TYPE elementStatus :
(
    Bad := 0,
    Timeout := 1,
	Unknown := 11,
    Good := 12
);
END_TYPE

(* stored: Version 1.1.0.1, ProductVersion 3.1.0.36
   DUT elementStatus: Id {b682ee42-3264-4a62-ad0c-29f8d3426a73} *)
